FUNCTION_BLOCK FB_ShippingRobot_Right EXTENDS FB_RobotRegionMove_BufferArea
VAR_INPUT
	Buzz	: REFERENCE TO BOOL;
	RedLamp	: REFERENCE TO BOOL;
	bCompleteRequest	: BOOL;
	Input		: REFERENCE TO ST_InputTable;
END_VAR
VAR_OUTPUT
	bTransCVInPosition : BOOL;
END_VAR
VAR
	//Area : E_RobotArea := E_RobotArea.TransmitCV_End;
	Blink		: ST_BlinkInfo;
	BuzzBlinker	: Blink;
	LightBlinker: Blink;
	TrigBuzz	: R_TRIG;
	TrigLight	: R_TRIG;
	BlinkInfo	: ST_BlinkInfo;
	
	TON_BlinkDelay	: TON;
END_VAR

SUPER^.A10_StateControl();
A00_BasicUnits();
Area := E_RobotArea.ShippingRobotRight;

ACTION A00_BasicUnits:
tonTimeOut(PT:=T#60S);
TON_BlinkDelay(PT:= T#1S);

bTransCVInPosition := Input.bShippingTransCV_Rightside_Arrived;
ErrorID:=2250;
END_ACTION

METHOD M_CheckCommand : BOOL // True : Command is useful
VAR_INPUT
END_VAR
VAR
	
END_VAR
// Check command paremeter is correct

THIS^.Get :=Info.Get;
UseA := Info.UseA;
UseB := Info.UseB;
//Buffer area
		
IF UseA AND ( Info.A_Position<1 OR  Info.A_Position>40) THEN
	strStatus:='Wrong command ,Position A Not allow';
	M_CheckCommand:=FALSE;
	RETURN;			
END_IF		

IF UseB AND( Info.B_Position<1 OR  Info.B_Position>40 )THEN
	strStatus:='Wrong command ,Position B Not allow';
	M_CheckCommand:=FALSE;
	RETURN;			
END_IF
		
IF Get THEN
	IF NOT Robot._DI1.ClampA_Open THEN
		strStatus := 'Get command , clamp have box ';
		M_CheckCommand := FALSE;
		RETURN;
	END_IF
ELSE
	IF Robot._DI1.ClampA_Open THEN 
		strStatus := 'Place command , clamp not have box ';
		M_CheckCommand := FALSE;
		RETURN;
	END_IF
END_IF
M_CheckCommand:=TRUE;
END_METHOD

METHOD M_CheckUnitsNotBusy : BOOL
VAR_INPUT
END_VAR
M_CheckUnitsNotBusy := true;
END_METHOD

METHOD M_CheckUnitsReady : BOOL
VAR_INPUT
END_VAR
M_CheckUnitsReady := true;
END_METHOD

METHOD  M_STATE_ABORTED
VAR_INPUT
END_VAR
ERROR :=TRUE;
Busy    := FALSE;
Aborted := TRUE;
Status := strStatus;
_AbortCompleted := FALSE;
uiAbortingStep := 0;
UniqueErrorCode:=_UniqueErrorCode;

IF NOT Execute THEN
	eSTATE:=STATE_RESETTING;
END_IF

IF Execute AND Reset THEN
		Error := FALSE;
	Aborted := false;
	uiExecutingStep :=uiResumeStep;
	PreviousStrStatus := strStatus;
	PreviousErrorCode := _UniqueErrorCode;

	eSTATE:=STATE_EXECUTING;
END_IF
END_METHOD

METHOD  M_STATE_ABORTING
VAR_INPUT
END_VAR
CASE uiAbortingStep OF
	0 :
		_Abort := FALSE;
		Abort 			:= false;
		uiAbortingStep:=9999;
		tonTimeOut.IN := FALSE;
		IF strStatus = PreviousStrStatus THEN
			_UniqueErrorCode :=PreviousErrorCode;
		END_IF
		_Abort :=FALSE;
	9999:	_AbortCompleted:=TRUE;
END_CASE

IF _AbortCompleted THEN	
	eSTATE :=STATE_ABORTED;
END_IF
END_METHOD

METHOD  M_STATE_DONE
VAR_INPUT
END_VAR
Busy := FALSE;
Done := TRUE;
IF NOT Execute THEN
    eState := STATE_RESETTING;
END_IF
END_METHOD

METHOD  M_STATE_DORMANT
VAR_INPUT
END_VAR
// Clear FB output
Busy            := FALSE;
Done            := FALSE;
Aborted         := FALSE;
Error           := FALSE;
ErrorID         := 0;
Status          := '';
_ResetCompleted := FALSE;
_Error          := FALSE;
_Executed       := FALSE;

bCompleteRequest := false;
TON_BlinkDelay.IN := FALSE;
tonTimeOut.IN:=FALSE;
strStatus :='No Error';
uiExecutingStep :=uiResettingStep :=uiResumeStep :=0;
PreviousStrStatus			 :='';
PreviousErrorCode			 :='';
_UniqueErrorCode	:='0';

// Wait Execute command
IF Execute AND bTransCVInPosition THEN
    eState := STATE_EXECUTING;
ELSE
	strStatus :='Wrong command ,TransCV not In Position ';
	_ERROR := TRUE;
END_IF
END_METHOD

METHOD  M_STATE_ERROR
VAR_INPUT
END_VAR
ERROR   :=TRUE;
Busy	:=FALSE;
Status := strStatus;
UniqueErrorCode:=_UniqueErrorCode;
IF NOT Execute THEN	
eSTATE:=STATE_RESETTING;
END_IF
END_METHOD

METHOD  M_STATE_EXECUTING
VAR_INPUT
END_VAR
VAR_INST
    ActionMode       : E_ReloadRoundBoxAction;
	BoxReady_1st : BOOL;
	BoxReady_2nd : BOOL;
    CarrierReady_1st : BOOL;
    CarrierReady_2nd : BOOL;
    uiBothStep : UINT;
    uiSingleClampStep : UINT;
	Address_A : INT;
	Address_B : INT;
END_VAR
VAR
	WareHouse: INT;
END_VAR
// Set Busy active edit by johnson
Busy := TRUE;
IF THIS^.Stop THEN // Pending the timeout when Stop signal occur
	tonTimeout.IN :=FALSE;
END_IF
// Service Process
CASE uiExecutingStep OF
	0:
        // Clear variable
        ActionMode       := E_ReloadRoundBoxAction.Undefined;
        CarrierReady_1st := FALSE;
        CarrierReady_2nd := FALSE;
        uiBothStep := 0;
		uiSingleClampStep :=0;
		BoxReady_1st := 0;
		BoxReady_2nd := 0;
		tonTimeOut.IN:=FALSE;
        // Check command
        IF M_CheckCommand() THEN
            uiExecutingStep := 10;
		ELSE
			_Error:=TRUE;
        END_IF
    10:
        // Start process, check units first
        IF M_CheckUnitsReady() THEN
            uiExecutingStep := 20;
        END_IF
    20:
        // CHeck units not busy state
        IF M_CheckUnitsNotBusy() THEN
            uiExecutingStep := 1000;
        END_IF
   
	1000:   
			// Read   coordinate
 			 Address_A := LREAL_TO_INT(Info.A_Position);
			 Address_B := LREAL_TO_INT(Info.B_Position);
			 
			IF UseA AND NOT UseB THEN
				//Only clampA
				uiExecutingStep := 10000;
			ELSIF NOT UseA AND UseB THEN
				//Only ClampB 
				uiExecutingStep := 20000;
			ELSIF UseA AND UseB THEN
				//Both Clamps
				uiExecutingStep := 30000;		
			END_IF
       
    10000: // Only ClampA 
        IF NOT Robot._DI1.Done THEN            
           		BoxReady_1st:=TRUE;				
			          		 
				  // Robot Abs move
           		 Robot.M_StartRobotAbsMove(GetBox:=Get,
											UseClampA:=UseA,
											UseClampB:=UseB,
											Area:=Area,
											ClampA_Address:=Address_A,
											ClampB_Address:=Address_B,
											BoxReady_1:=BoxReady_1st,
											BoxReady_2:=BoxReady_2nd);	  
		
        ELSE
			tonTimeOut.IN:=FALSE;
            uiExecutingStep := 10080;
        END_IF
		tonTimeOut.IN:=TRUE;
		IF tonTimeOut.Q=TRUE THEN
			tonTimeOut.IN:=FALSE;			
			strStatus :='Action Robot timeout';
			_Abort:=TRUE;
			uiResettingStep := 10000;
		END_IF	
		IF Robot.Error THEN
			_Abort := TRUE;
			strStatus := 'FB_ShippingRobot place box to right Plate , Robot Error';
			uiResettingStep := 10000;
		END_IF
		
    10080:
        Robot.M_ResetRobotAbsMove(UseA,UseB); // Clear command and go to place box
		tonTimeOut.IN:=TRUE;
        IF NOT Robot._DI1.Done THEN
			tonTimeOut.IN:=FALSE;
            uiExecutingStep := 90000; 
        END_IF
    	IF tonTimeOut.Q=TRUE THEN
			strStatus :='Reset Robot timeout';
			uiResettingStep := 10080;
			_Abort:=TRUE;
		END_IF	
    
   20000: // Only ClampB
        IF NOT Robot._DI1.Done THEN           		
				BoxReady_2nd:=TRUE;				          		 
				  // Robot Abs move
           		 Robot.M_StartRobotAbsMove( GetBox:=Get,
											UseClampA:=UseA,
											UseClampB:=UseB,
											Area:=Area,
											ClampA_Address:=Address_A,
											ClampB_Address:=Address_B,
											BoxReady_1:=BoxReady_1st,
											BoxReady_2:=BoxReady_2nd);	
        ELSE
			tonTimeOut.IN:=FALSE;
            uiExecutingStep := 20080;
        END_IF
		tonTimeOut.IN:=TRUE;
			IF tonTimeOut.Q=TRUE THEN
				tonTimeOut.IN:=FALSE;			
				strStatus :='Reset Robot timeout';
				_Error:=TRUE;
			END_IF	
    20080:
       Robot.M_ResetRobotAbsMove(UseA,UseB);; // Clear command 

        IF NOT Robot._DI1.Done THEN
            uiExecutingStep := 90000; 
        END_IF
		tonTimeOut.IN:=TRUE;
		IF tonTimeOut.Q=TRUE THEN
			strStatus :='Reset Robot timeout';
			_Error:=TRUE;
		END_IF	
    30000: // Both Clamps
        		
		
		  CASE uiBothStep OF
           		0://	
					BoxReady_1st := FALSE;
					BoxReady_2nd := FALSE;					
					uiBothStep:=1000;	
	
				1000:
						BoxReady_1st:=TRUE;
						uiBothStep:=2000;
						
				2000:
						IF Robot._DI1.Notification THEN
							uiBothStep:=3000;
						END_IF
				3000:
					
					
						uiBothStep:=9000;	
					
				9000:
						BoxReady_2nd:=TRUE;
						uiBothStep:=9999;
				
				9999: //Wait		
        // wait reset
        END_CASE

       	  // Robot Abs move
           		 Robot.M_StartRobotAbsMove( GetBox:=Get,
											UseClampA:=UseA,
											UseClampB:=UseB,
											Area:=Area,
											ClampA_Address:=Address_A,
											ClampB_Address:=Address_B,
											BoxReady_1:=BoxReady_1st,
											BoxReady_2:=BoxReady_2nd);	
		
		
        IF Robot._DI1.Done THEN
			tonTimeOut.IN:=FALSE;
            uiExecutingStep := 30080;
        END_IF
		IF tonTimeOut.Q=TRUE THEN
				tonTimeOut.IN:=FALSE;			
				strStatus :='Reset Robot timeout';
				_Error:=TRUE;
			END_IF	
    30080: // Check robot command is clear
        
        Robot.M_ResetRobotAbsMove(UseA,UseB);

        IF NOT Robot._DI1.Done THEN
			tonTimeOut.IN:=FALSE;
            uiExecutingStep := 90000; // go to place step
        END_IF    
   		tonTimeOut.IN:=TRUE;
		IF tonTimeOut.Q=TRUE THEN
			strStatus :='Stop Robot timeout';
			_Error:=TRUE;
		END_IF	
   
	90000:
			IF bCompleteRequest THEN
				uiExecutingStep := 91000;
			ELSE
				uiExecutingStep := 99000;
			END_IF
			
	91000:	// shipping allocate mission complete signal
		BuzzBlinker(ENABLE:=TRUE , TIMELOW:=T#0.3S , TIMEHIGH:=T#0.3S , OUT=> Buzz);
		LightBlinker(ENABLE := TRUE , TIMELOW := T#0.3S , TIMEHIGH := T#0.3S , OUT => RedLamp );
		TrigBuzz(CLK:=Buzz);
		TrigLight(CLK :=RedLamp);
		IF TrigBuzz.Q THEN
			BlinkInfo.BuzzCount := BlinkInfo.BuzzCount +1;
		END_IF
		IF TrigLight.Q THEN
			BlinkInfo.LightCount := BlinkInfo.LightCount +1;
		END_IF
		
		IF BlinkInfo.BuzzCount >= BlinkInfo.MaxBuzzCOunt AND BlinkInfo.LightCount >=BlinkInfo.MaxLightCount THEN
			TON_BlinkDelay.IN :=TRUE;
			IF TON_BlinkDelay.q THEN
				uiExecutingStep := 99000;
			END_IF
		END_IF
   
		
    99000: // process done
		TON_BlinkDelay.IN := FALSE;
        Status    := 'Process completed';
        _Executed := TRUE;
END_CASE

IF _Executed THEN
    eState := STATE_DONE;
ELSIF _Error THEN
	//FUN_UniqueErrorCodeGenerator(iErrorID := ErrorID,UinqueErrorCode=>_UniqueErrorCode);
    eState := STATE_ERROR;
ELSIF NOT Execute THEN
    eState := STATE_RESETTING;
END_IF
IF _Abort OR Abort THEN
	//FUN_UniqueErrorCodeGenerator(iErrorID := ErrorID,UinqueErrorCode=>_UniqueErrorCode);
	eSTATE:=STATE_ABORTING;
END_IF
END_METHOD

METHOD  M_STATE_RESETTING
VAR_INPUT
END_VAR
Error :=FALSE;
Done :=FALSE;
Busy := FALSE;


CASE uiResettingStep OF
	
	0:
		bCompleteRequest := false;
		TON_BlinkDelay.IN := FALSE;
		tonTimeOut.IN:=FALSE;
		//Robot.M_ResetAllCommand();
		Robot.M_ResetRobotAbsMove(TRUE,TRUE);
		
		uiResettingStep:=9999;
	9999:
		_ResetCompleted:=TRUE;
END_CASE
IF _ResetCompleted THEN
	eSTATE:=STATE_DORMANT;
END_IF
END_METHOD

END_FUNCTION_BLOCK

(* stored: Version 1.1.0.1, ProductVersion 3.1.4024.13
   POU FB_ShippingRobot_Right: Id {ee609f86-085a-4b67-a9a8-7bedfbb17379}, SpecialFunc None
   Folder Method: Id {4d645e10-235d-4329-bbe3-140b43c019ec}
   Folder State: Id {a4c10a5f-e8d1-4a85-a4ae-cb6fe648f92e}
   Action A00_BasicUnits: Id {4eacd091-9963-40d2-be0d-0c029e90a68a}
   Method M_CheckCommand: Id {42e9c988-6627-48ce-bb4d-909e434a05ed}
   Method M_CheckUnitsNotBusy: Id {1732ba49-846a-47c8-aae3-645eda5346ea}
   Method M_CheckUnitsReady: Id {98f007bb-ac32-4061-91c0-215ffccf16ea}
   Method M_STATE_ABORTED: Id {a348bdc5-cc0d-48ea-a0bf-8b915fde8194}
   Method M_STATE_ABORTING: Id {e45f0efa-23b4-4d2f-a420-e9ea18b7a291}
   Method M_STATE_DONE: Id {cad33853-f2f8-4893-93fb-e7eb2f1ce3e3}
   Method M_STATE_DORMANT: Id {66f0e90c-9d44-4afb-867c-6f66bcd7b663}
   Method M_STATE_ERROR: Id {6bf1d6b6-f1ce-4753-bb84-a2b7874c9b01}
   Method M_STATE_EXECUTING: Id {86f80632-2070-4444-96e9-79455d36340d}
   Method M_STATE_RESETTING: Id {1e8dab63-8550-4fa6-befe-282584f514e7} *)
